Universal Robots PolyScope program: Subprogram1a.urp

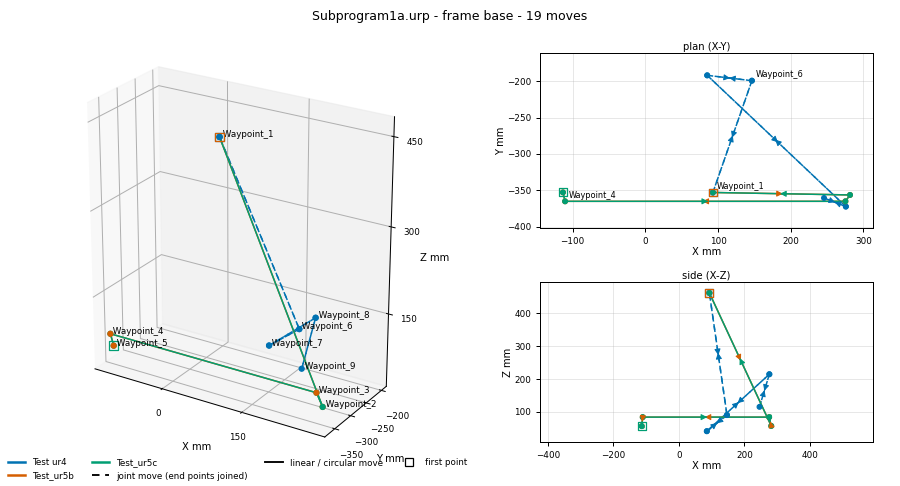
[picture p0: tool path of Subprogram1a.urp in frame base, 19 of 19 moves have a stored position in this frame; points joined in program order, loops and branches not executed]
Program PythonSubprogram1a (installation=default directory=/programs/usbdisk/NoodleBotSoftware createdIn=3.12.1.90940 lastSavedIn=3.12.1.90940 robotSerialNumber=2017354841)
Calibrated DH parameters: a=[0.000094, -0.006117, -0.382762, 0.000086, 0.000044, 0]; d=[0.089236, 217.751846, -204.357806, -13.283746, 0.094902, 0.082641]; alpha=[1.57017, 0.001953, -0.006493, 1.570192, -1.570543, 0]; deltaTheta=[0.000036, 1.556386, -1.779789, 0.223359, -0.000014, -0.000001]
BeforeStart
  var_1 := socket_open("192.168.0.100",30000)
Robot Program (runOnlyOnce=false)
  Loop While (checkContinuously=false) expression=var_1≟ False
    var_1 := socket_open("192.168.0.100",30000)
    Wait Sleep waitTime=0.5
  Script: socket_send_string("asking_for_data")
  Wait Sleep waitTime=0.5
  var_2 := socket_read_ascii_float(3)
  Wait Sleep waitTime=0.5
  var_1 := False
  If var_2[1]≟1
    Call Test ur4
  If var_2[1]≟1
    Call Test_ur5b
  If var_2[2]≟1 and digital_in[0]≟ False
    Set DigitalOutput pin=digital_out[4]; digitalValue=1
    Wait Sleep waitTime=3
    Set DigitalOutput pin=digital_out[4]; digitalValue=0
    Wait Sleep waitTime=0.5
    Set DigitalOutput pin=digital_out[5]; digitalValue=1
    Wait Sleep waitTime=3
    Set DigitalOutput pin=digital_out[5]; digitalValue=0
    Wait Sleep waitTime=0.5
  If var_2[3]≟1 and digital_in[0]≟ False
    Set DigitalOutput pin=digital_out[6]; digitalValue=1
    Wait Sleep waitTime=0.5
    Set DigitalOutput pin=digital_out[6]; digitalValue=0
    Wait Sleep waitTime=0.5
    Set DigitalOutput pin=digital_out[7]; digitalValue=1
    Wait Sleep waitTime=0.5
    Set DigitalOutput pin=digital_out[7]; digitalValue=0
    Wait Sleep waitTime=0.5
  If digital_in[0]≟ False
    Call Test_ur5c
    Wait Sleep waitTime=0.5
    var_1 := False
  Script: socket_close()
SubProgram -> Test ur4
SubProgram -> Test_ur5c
SubProgram -> Test_ur5b
SubProgram Test ur4 (keepSynchronizedWithDisk=false) programFile=/programs/Test ur4.urp
  MoveJ speed 120 deg/s, acceleration 90 deg/s^2 (useActiveTCP=true)
    URCap RG2 (RG - On Robot, OnRobot A/S) dataModel(depthCompensate=false, force=40, payload=0.0, width=50, name=RG2(50))
    Waypoint Waypoint_1: TCP in base x=92.939 y=-353.097 z=462.595 mm, rx=1.1692 ry=-1.2408 rz=1.1709 rad; joints [88.542, -137.018, 138.65, 178.588, 268.341, 89.999] deg; flange x=103.097 y=-166.778 z=463.297 mm, rx=1.2543 ry=1.1818 rz=-1.2438 rad
    Wait Sleep waitTime=1
    Waypoint Waypoint_6: TCP in base x=146.59 y=-199.362 z=90.11 mm, rx=-2.576 ry=0.0709 rz=1.786 rad; joints [138.196, -78.978, 116.17, 296.94, 232.836, 75.177] deg; flange x=321.213 y=-205.121 z=155.617 mm, rx=-0.0531 ry=-1.9288 rz=-0.0072 rad
    Wait Sleep waitTime=1
    Waypoint Waypoint_7: TCP in base x=85.124 y=-191.999 z=40.975 mm, rx=-2.2271 ry=-0.0602 rz=2.1803 rad; joints [135.848, -65.281, 123.713, 300.083, 225.086, 86.563] deg; flange x=271.64 y=-190.189 z=44.971 mm, rx=0.0431 ry=-1.5917 rz=-0.0272 rad
    URCap RG2 (RG - On Robot, OnRobot A/S) dataModel(depthCompensate=false, force=40, payload=0.0, width=0, name=RG2(0))
    Wait Sleep waitTime=1
    Waypoint Waypoint_8: TCP in base x=275.796 y=-372.44 z=214.652 mm, rx=1.4266 ry=0.952 rz=-1.4093 rad; joints [144.954, -87.311, 121.008, 317.01, 162.877, 85.328] deg; flange x=334.168 y=-195.422 z=206.762 mm, rx=0.9022 ry=-1.3519 rz=1.0444 rad
    Wait Sleep waitTime=1
    Waypoint Waypoint_9: TCP in base x=245.781 y=-360.651 z=115.199 mm, rx=1.0638 ry=-1.1694 rz=0.6215 rad; joints [144.976, -77.022, 127.234, 300.679, 169.785, 241.281] deg; flange x=324.968 y=-191.791 z=110.822 mm, rx=1.3897 ry=1.2641 rz=-1.7757 rad
    Wait Sleep waitTime=1
    Waypoint Waypoint_10: TCP in base x=275.796 y=-372.44 z=214.652 mm, rx=1.4266 ry=0.952 rz=-1.4093 rad; joints [144.954, -87.311, 121.008, 317.01, 162.877, 85.328] deg; flange x=334.168 y=-195.422 z=206.762 mm, rx=0.9022 ry=-1.3519 rz=1.0444 rad
    Wait Sleep waitTime=1
    Waypoint Waypoint_11: TCP in base x=85.124 y=-191.999 z=40.975 mm, rx=-2.2271 ry=-0.0602 rz=2.1803 rad; joints [135.848, -65.281, 123.713, 300.083, 225.086, 86.563] deg; flange x=271.64 y=-190.189 z=44.971 mm, rx=0.0431 ry=-1.5917 rz=-0.0272 rad
    URCap RG2 (RG - On Robot, OnRobot A/S) dataModel(depthCompensate=false, force=40, payload=0.0, width=50, name=RG2(50))
    Wait Sleep waitTime=1
    Waypoint Waypoint_12: TCP in base x=146.59 y=-199.362 z=90.11 mm, rx=-2.576 ry=0.0709 rz=1.786 rad; joints [138.196, -78.978, 116.17, 296.94, 232.836, 75.177] deg; flange x=321.213 y=-205.121 z=155.617 mm, rx=-0.0531 ry=-1.9288 rz=-0.0072 rad
    Wait Sleep waitTime=1
    Waypoint Waypoint_1: TCP in base x=92.939 y=-353.097 z=462.595 mm, rx=1.1692 ry=-1.2408 rz=1.1709 rad; joints [88.542, -137.018, 138.65, 178.588, 268.341, 89.999] deg; flange x=103.097 y=-166.778 z=463.297 mm, rx=1.2543 ry=1.1818 rz=-1.2438 rad
    Wait Sleep waitTime=1
SubProgram Test_ur5b (keepSynchronizedWithDisk=false) programFile=/programs/Test ur5b.urp
  MoveL speed 1000 mm/s, acceleration 1200 mm/s^2 (useActiveTCP=true) feature=Base
    URCap RG2 (RG - On Robot, OnRobot A/S) dataModel(depthCompensate=false, force=40, payload=0.0, width=85, name=RG2(85))
    Waypoint Waypoint_1: TCP in base x=92.939 y=-353.097 z=462.595 mm, rx=1.1692 ry=-1.2408 rz=1.1709 rad; joints [88.542, -137.018, 138.65, 178.588, 268.341, 89.999] deg; flange x=103.097 y=-166.778 z=463.297 mm, rx=1.2543 ry=1.1818 rz=-1.2438 rad
    Wait Sleep waitTime=0.1
    Waypoint Waypoint_2: TCP in base x=281.568 y=-356.493 z=57.062 mm, rx=2.4509 ry=-1.0812 rz=-0.3973 rad; joints [131.142, -83.255, 116.241, 241.937, 240.139, 90.003] deg; flange x=360.116 y=-306.414 z=218.729 mm, rx=-1.1245 ry=-2.5488 rz=0.6202 rad
    URCap RG2 (RG - On Robot, OnRobot A/S) dataModel(depthCompensate=false, payload=0.0, force=40, width=0, name=RG2(0))
    Wait Sleep waitTime=0.1
    Waypoint Waypoint_3: TCP in base x=275.23 y=-365.244 z=83.858 mm, rx=2.4082 ry=-1.0628 rz=-0.4074 rad; joints [131.131, -84.8, 114.576, 244.685, 237.533, 90.016] deg; flange x=358.189 y=-309.185 z=241.34 mm, rx=-1.1149 ry=-2.5256 rz=0.6807 rad
    Wait Sleep waitTime=0.1
    Waypoint Waypoint_4: TCP in base x=-110.35 y=-365.263 z=83.889 mm, rx=2.4083 ry=-1.0627 rz=-0.4074 rad; joints [69.173, -109.993, 144.496, 207.947, 251.859, 22.112] deg; flange x=-27.414 y=-309.154 z=241.302 mm, rx=-1.1146 ry=-2.5256 rz=0.6805 rad
    Wait Sleep waitTime=0.1
    Waypoint Waypoint_5: TCP in base x=-113.251 y=-352.97 z=56.401 mm, rx=2.4743 ry=-1.0833 rz=-0.4569 rad; joints [69.146, -107.002, 145.454, 208.35, 250.31, 22.145] deg; flange x=-30.387 y=-310.642 z=218.159 mm, rx=-1.1049 ry=-2.5237 rz=0.5697 rad
    Wait Sleep waitTime=0.1
SubProgram Test_ur5c (keepSynchronizedWithDisk=false) programFile=/programs/Test ur5c.urp
  MoveL speed 1000 mm/s, acceleration 1200 mm/s^2 (useActiveTCP=true) feature=Base
    Waypoint Waypoint_5: TCP in base x=-113.251 y=-352.97 z=56.401 mm, rx=2.4743 ry=-1.0833 rz=-0.4569 rad; joints [69.146, -107.002, 145.454, 208.35, 250.31, 22.145] deg; flange x=-30.387 y=-310.642 z=218.159 mm, rx=-1.1049 ry=-2.5237 rz=0.5697 rad
    Wait Sleep waitTime=0.1
    Waypoint Waypoint_4: TCP in base x=-110.35 y=-365.263 z=83.889 mm, rx=2.4083 ry=-1.0627 rz=-0.4074 rad; joints [69.173, -109.993, 144.496, 207.947, 251.859, 22.112] deg; flange x=-27.414 y=-309.154 z=241.302 mm, rx=-1.1146 ry=-2.5256 rz=0.6805 rad
    Wait Sleep waitTime=0.1
    Waypoint Waypoint_3: TCP in base x=275.23 y=-365.244 z=83.858 mm, rx=2.4082 ry=-1.0628 rz=-0.4074 rad; joints [131.131, -84.8, 114.576, 244.685, 237.533, 90.016] deg; flange x=358.189 y=-309.185 z=241.34 mm, rx=-1.1149 ry=-2.5256 rz=0.6807 rad
    Wait Sleep waitTime=0.1
    Waypoint Waypoint_2: TCP in base x=281.568 y=-356.493 z=57.062 mm, rx=2.4509 ry=-1.0812 rz=-0.3973 rad; joints [131.142, -83.255, 116.241, 241.937, 240.139, 90.003] deg; flange x=360.116 y=-306.414 z=218.729 mm, rx=-1.1245 ry=-2.5488 rz=0.6202 rad
    URCap RG2 (RG - On Robot, OnRobot A/S) dataModel(depthCompensate=false, force=40, payload=0.0, width=85, name=RG2(85))
    Wait Sleep waitTime=0.1
    Waypoint Waypoint_1: TCP in base x=92.939 y=-353.097 z=462.595 mm, rx=1.1692 ry=-1.2408 rz=1.1709 rad; joints [88.542, -137.018, 138.65, 178.588, 268.341, 89.999] deg; flange x=103.097 y=-166.778 z=463.297 mm, rx=1.2543 ry=1.1818 rz=-1.2438 rad
    Wait Sleep waitTime=0.1
